// TIA Portal V17 export
// export: Created 2023-05-07T12:12:23.0129328Z, ExportSetting WithDefaults, DisplayName Totally Integrated Automation Portal, DisplayVersion V17, DisplayName TIA Portal Openness, DisplayVersion V17, DisplayName TIA Portal Version Control Interface, DisplayVersion V17, DisplayName TIA Portal Test Suite Advanced, DisplayVersion V17, DisplayName STEP 7 Professional, DisplayVersion V17, DisplayName SIMATIC Energy Suite, DisplayVersion V17, DisplayName STEP 7 Safety, DisplayVersion V17, DisplayName WinCC Professional, DisplayVersion V17
DATA_BLOCK "Inversion_DB"   // DB17
VERSION : 0.1
// stored: AutoNumber true, InstanceOfName Inversion, InstanceOfType FB
"Inversion"
   // VAR_INPUT
   //    wejscie : Real;
   // END_VAR
   // VAR_OUTPUT
   //    wyjscie : Real;
   // END_VAR
   // VAR
   //    x : Array[0..5] of Real;
   //    s : Array[0..7] of Real;
   //    o : Array[0..7] of Real;
   //    s2 : Real;
   //    i : Int;
   //    w1_1 : Array[0..7] of Real;
   //    w1_2 : Array[0..7] of Real;
   //    w1_3 : Array[0..7] of Real;
   //    w1_4 : Array[0..7] of Real;
   //    w1_5 : Array[0..7] of Real;
   //    w1_6 : Array[0..7] of Real;
   //    w_2 : Array[0..7] of Real;
   //    bias : Array[0..7] of Real;
   //    bias2 : Real;
   //    N : Int;
   // END_VAR
BEGIN
END_DATA_BLOCK
